	(* Internal method *)
	{attribute 'hide'}
	METHOD FB_init : BOOL
	VAR_INPUT
		(*  if TRUE, the retain variables are initialized (warm start / cold start) *)
		bInitRetains : BOOL;
		(*  if TRUE, the instance afterwards gets moved into the copy code (online change) *)
		bInCopyCode : BOOL;
	END_VAR
END_METHOD


	(* Internal method *)
	{attribute 'hide'}
	METHOD FB_exit : BOOL
	VAR_INPUT
		(*  if TRUE, the exit method is called for exiting an instance that is copied afterwards (online change). *)
		bInCopyCode : BOOL;
	END_VAR
END_METHOD


	(* Set the rotation angle in degrees [Â°]. *)
	METHOD SetAngle
	VAR_INPUT
		(* Rotation angle to set in degrees [Â°]. *)
		angle : LREAL;
	END_VAR
END_METHOD


	(* Set the components of this vector to '0.0'. *)
	METHOD SetZero
END_METHOD


	(* Set the components of this orientation. *)
	METHOD SetValues
	VAR_IN_OUT
		(* The position values to set. *)
 {attribute 'GUID' := '86B4AC92-A3FD-99C6-DFBE-A266E31A06E2'}
				orientation2D : Orientation2D;
	END_VAR
END_METHOD


	(* Get the direction of the local x-axis. *)
	METHOD GetDirectionX
	VAR_IN_OUT
		(* The local x-direction of this orientation. *)
 {attribute 'GUID' := '4CE6AEBB-A122-94B9-C485-29D927BD5C71'}
				localX : TangentXY;
	END_VAR
END_METHOD


	(* Get the direction of the local y-axis. *)
	METHOD GetDirectionY
	VAR_IN_OUT
		(* The local y-direction of this orientation. *)
 {attribute 'GUID' := '4CE6AEBB-A122-94B9-C485-29D927BD5C71'}
				localY : TangentXY;
	END_VAR
END_METHOD


	(* Invert this position. *)
	METHOD Invert
END_METHOD


	(* Multiply an orientation to this orientation. *)
	METHOD ConcatenateWith
	VAR_IN_OUT
		(* Orientation to concatenate with. *)
 {attribute 'GUID' := '86B4AC92-A3FD-99C6-DFBE-A266E31A06E2'}
				orientation2D : Orientation2D;
	END_VAR
END_METHOD


	(* Turn the orientation. *)
	METHOD TurnByC
	VAR_INPUT
		(* Rotation angle to turn by in degrees [Â°]. *)
		angle : LREAL;
	END_VAR
END_METHOD


	(* Rotate a PositionXY according to this orientation. *)
	METHOD Transform
	VAR_IN_OUT
		(* The orientation to multipy by. *)
 {attribute 'GUID' := 'FCACA74E-C57F-9E9F-C3FF-7BECD9A9CD0E'}
				positionXY : PositionXY;
	END_VAR
END_METHOD


	PROPERTY angle : LREAL
GET
END_GET
SET
END_SET
END_PROPERTY

END_FUNCTION_BLOCK

// POUs/Spatial/Functions/ConcatenateABC

	{attribute 'TcIecLibraryType'}
	{attribute 'external_name' := 'ConcatenateABC_GUID_72325069_8572_94A4_CBCD_8734C10F3E88'}
	(* Concatenate two instances of Orientation3D. *)
	FUNCTION ConcatenateABC : BOOL
	VAR_IN_OUT
		rotation0	:	Orientation3D;	(* 1st input orientation of the concatenation. *)
		rotation1	:	Orientation3D;	(* 2nd input orientation of the concatenation. *)
		concatenation	:	Orientation3D;	(* The concatenation of the two input instances. *)
	END_VAR

END_FUNCTION

// POUs/Spatial/Positions/Orientation3D

	{attribute 'c++_compatible'}
	{attribute 'external_name' := 'Orientation3D_GUID_E2786DA7_805D_90A4_CCD0_35D19D53662E'}
	{attribute 'TcIecLibraryType'}
	{attribute 'no_explicit_call' :='do not call this POU directly'}
	{attribute 'no_assign'}
	(* 3D orientation. All angles in degrees [Â°]. *)
	FUNCTION_BLOCK Orientation3D
	VAR
		(* Rotation around the 1st local axis in degrees [Â°]. *)
		p0 : LREAL;
		(* Rotation around 2nd local axis in degrees [Â°]. *)
		p1 : LREAL;
		(* Rotation around 3rd local axis in degrees [Â°]. *)
		p2 : LREAL;
		(* Defines the rotation order (rotate around local axes from left to right) *)
		 {attribute 'GUID' := 'BF8BCC1E-925E-4A57-801C-CC42AFDDA86D'}
		coordinates : E_RotationCoordinates := E_RotationCoordinates.CBA;
		 {attribute 'hide'}
		_reserved1 : ARRAY [1..84] OF USINT;
	END_VAR


	(* Internal method *)
	{attribute 'hide'}
	METHOD FB_init : BOOL
	VAR_INPUT
		(*  if TRUE, the retain variables are initialized (warm start / cold start) *)
		bInitRetains : BOOL;
		(*  if TRUE, the instance afterwards gets moved into the copy code (online change) *)
		bInCopyCode : BOOL;
	END_VAR
END_METHOD


	(* Internal method *)
	{attribute 'hide'}
	METHOD FB_exit : BOOL
	VAR_INPUT
		(*  if TRUE, the exit method is called for exiting an instance that is copied afterwards (online change). *)
		bInCopyCode : BOOL;
	END_VAR
END_METHOD


	(* Set the components of this vector to '0.0'. *)
	METHOD SetZero
END_METHOD


	(* Set the components of this position. *)
	METHOD SetValues
	VAR_IN_OUT
		(* The position values to set. *)
 {attribute 'GUID' := 'E2786DA7-805D-90A4-CCD0-35D19D53662E'}
				orientation3D : Orientation3D;
	END_VAR
END_METHOD


	(* Set the coordinates of the orientation. *)
	METHOD SetValuesABC
	VAR_INPUT
		(* 1st rotation angle in degrees [Â°]. *)
		phi0 : LREAL;
		(* 2nd rotation angle in degrees [Â°]. *)
		phi1 : LREAL;
		(* 3rd rotation angle in degrees [Â°]. *)
		phi2 : LREAL;
	END_VAR
END_METHOD


	(* Set the coordinates of the orientation. *)
	METHOD SetValuesACB
	VAR_INPUT
		(* 1st rotation angle in degrees [Â°]. *)
		phi0 : LREAL;
		(* 2nd rotation angle in degrees [Â°]. *)
		phi1 : LREAL;
		(* 3rd rotation angle in degrees [Â°]. *)
		phi2 : LREAL;
	END_VAR
END_METHOD


	(* Set the coordinates of the orientation. *)
	METHOD SetValuesBCA
	VAR_INPUT
		(* 1st rotation angle in degrees [Â°]. *)
		phi0 : LREAL;
		(* 2nd rotation angle in degrees [Â°]. *)
		phi1 : LREAL;
		(* 3rd rotation angle in degrees [Â°]. *)
		phi2 : LREAL;
	END_VAR
END_METHOD


	(* Set the coordinates of the orientation. *)
	METHOD SetValuesBAC
	VAR_INPUT
		(* 1st rotation angle in degrees [Â°]. *)
		phi0 : LREAL;
		(* 2nd rotation angle in degrees [Â°]. *)
		phi1 : LREAL;
		(* 3rd rotation angle in degrees [Â°]. *)
		phi2 : LREAL;
	END_VAR
END_METHOD


	(* Set the coordinates of the orientation. *)
	METHOD SetValuesCAB
	VAR_INPUT
		(* 1st rotation angle in degrees [Â°]. *)
		phi0 : LREAL;
		(* 2nd rotation angle in degrees [Â°]. *)
		phi1 : LREAL;
		(* 3rd rotation angle in degrees [Â°]. *)
		phi2 : LREAL;
	END_VAR
END_METHOD


	(* Set the coordinates of the orientation. *)
	METHOD SetValuesCBA
	VAR_INPUT
		(* 1st rotation angle in degrees [Â°]. *)
		phi0 : LREAL;
		(* 2nd rotation angle in degrees [Â°]. *)
		phi1 : LREAL;
		(* 3rd rotation angle in degrees [Â°]. *)
		phi2 : LREAL;
	END_VAR
END_METHOD


	(* Set the coordinates of the orientation. *)
	METHOD SetValuesABA
	VAR_INPUT
		(* 1st rotation angle in degrees [Â°]. *)
		phi0 : LREAL;
		(* 2nd rotation angle in degrees [Â°]. *)
		phi1 : LREAL;
		(* 3rd rotation angle in degrees [Â°]. *)
		phi2 : LREAL;
	END_VAR
END_METHOD


	(* Set the coordinates of the orientation. *)
	METHOD SetValuesACA
	VAR_INPUT
		(* 1st rotation angle in degrees [Â°]. *)
		phi0 : LREAL;
		(* 2nd rotation angle in degrees [Â°]. *)
		phi1 : LREAL;
		(* 3rd rotation angle in degrees [Â°]. *)
		phi2 : LREAL;
	END_VAR
END_METHOD


	(* Set the coordinates of the orientation. *)
	METHOD SetValuesBCB
	VAR_INPUT
		(* 1st rotation angle in degrees [Â°]. *)
		phi0 : LREAL;
		(* 2nd rotation angle in degrees [Â°]. *)
		phi1 : LREAL;
		(* 3rd rotation angle in degrees [Â°]. *)
		phi2 : LREAL;
	END_VAR
END_METHOD


	(* Set the coordinates of the orientation. *)
	METHOD SetValuesBAB
	VAR_INPUT
		(* 1st rotation angle in degrees [Â°]. *)
		phi0 : LREAL;
		(* 2nd rotation angle in degrees [Â°]. *)
		phi1 : LREAL;
		(* 3rd rotation angle in degrees [Â°]. *)
		phi2 : LREAL;
	END_VAR
END_METHOD


	(* Set the coordinates of the orientation. *)
	METHOD SetValuesCAC
	VAR_INPUT
		(* 1st rotation angle in degrees [Â°]. *)
		phi0 : LREAL;
		(* 2nd rotation angle in degrees [Â°]. *)
		phi1 : LREAL;
		(* 3rd rotation angle in degrees [Â°]. *)
		phi2 : LREAL;
	END_VAR
END_METHOD


	(* Set the coordinates of the orientation. *)
	METHOD SetValuesCBC
	VAR_INPUT
		(* 1st rotation angle in degrees [Â°]. *)
		phi0 : LREAL;
		(* 2nd rotation angle in degrees [Â°]. *)
		phi1 : LREAL;
		(* 3rd rotation angle in degrees [Â°]. *)
		phi2 : LREAL;
	END_VAR
END_METHOD


	(* Get the direction of the local x-axis. *)
	METHOD GetDirectionX
	VAR_IN_OUT
		(* The local x-direction of this orientation. *)
 {attribute 'GUID' := '9F987066-55C3-9A71-FEA1-9CB49A451CD6'}
				localX : Tangent3D;
	END_VAR
END_METHOD


	(* Get the direction of the local y-axis. *)
	METHOD GetDirectionY
	VAR_IN_OUT
		(* The local y-direction of this orientation. *)
 {attribute 'GUID' := '9F987066-55C3-9A71-FEA1-9CB49A451CD6'}
				localY : Tangent3D;
	END_VAR
END_METHOD


	(* Get the direction of the local z-axis. *)
	METHOD GetDirectionZ
	VAR_IN_OUT
		(* The local z-direction of this orientation. *)
 {attribute 'GUID' := '9F987066-55C3-9A71-FEA1-9CB49A451CD6'}
				localZ : Tangent3D;
	END_VAR
END_METHOD


	(* Invert this position. *)
	METHOD Invert
END_METHOD


	(* Multiply an orientation to this orientation. *)
	METHOD ConcatenateWith
	VAR_IN_OUT
		(* Orientation to concatenate with. *)
 {attribute 'GUID' := 'E2786DA7-805D-90A4-CCD0-35D19D53662E'}
				orientation : Orientation3D;
	END_VAR
END_METHOD


	(* Rotate around an arbitrary local axis. The turn angle is given by the length of the axis. *)
	METHOD TurnBy
	VAR_IN_OUT
		(* The axis of rotation. Its length represents the angle of rotation in degrees [Â°]. *)
 {attribute 'GUID' := '6DC08058-799F-98C7-C4DD-73FA46FCF197'}
				axis : TangentABC;
	END_VAR
END_METHOD


	(* Rotation around the local x-axis. *)
	METHOD TurnByA
	VAR_INPUT
		(* The angle to rotate by in degrees [Â°]. *)
		da : LREAL;
	END_VAR
END_METHOD


	(* Rotation around the local y-axis. *)
	METHOD TurnByB
	VAR_INPUT
		(* The angle to rotate by in degrees [Â°]. *)
		db : LREAL;
	END_VAR
END_METHOD


	(* Rotation around the local z-axis. *)
	METHOD TurnByC
	VAR_INPUT
		(* The angle to rotate by in degrees [Â°]. *)
		dc : LREAL;
	END_VAR
END_METHOD


	(* Rotate a Position3D according to this orientation. *)
	METHOD Transform
	VAR_IN_OUT
		(* Position to transform. *)
 {attribute 'GUID' := '40E6105C-AAE1-907F-E93C-27FE8D6C7544'}
				position3D : Position3D;
	END_VAR
END_METHOD


	PROPERTY phi0 : LREAL
GET
END_GET
SET
END_SET
END_PROPERTY


	PROPERTY phi1 : LREAL
GET
END_GET
SET
END_SET
END_PROPERTY


	PROPERTY phi2 : LREAL
GET
END_GET
SET
END_SET
END_PROPERTY


	PROPERTY convention : E_RotationCoordinates
GET
END_GET
SET
END_SET
END_PROPERTY

END_FUNCTION_BLOCK

// POUs/Spatial/Functions/ConcatenateXYC

	{attribute 'TcIecLibraryType'}
	{attribute 'external_name' := 'ConcatenateXYC_GUID_55AD0630_DF53_9402_CBF6_9E8FF05A606D'}
	(* Concatenate two instances of PositionXYC. *)
	FUNCTION ConcatenateXYC : BOOL
	VAR_IN_OUT
		position0	:	PositionXYC;	(* 1st input position of the concatenation. *)
		position1	:	PositionXYC;	(* 2nd input position of the concatenation. *)
		concatenation	:	PositionXYC;	(* The concatenation of the two input instances. *)
	END_VAR

END_FUNCTION

// POUs/Spatial/Functions/Concatenate6D

	{attribute 'TcIecLibraryType'}
	{attribute 'external_name' := 'Concatenate6D_GUID_A3C51CBA_D129_9074_F963_7F4312C3BE5C'}
	(* Concatenate two instances of PositionSE3. *)
	FUNCTION Concatenate6D : BOOL
	VAR_IN_OUT
		position0	:	PositionSE3;	(* 1st input position of the concatenation. *)
		position1	:	PositionSE3;	(* 2nd input position of the concatenation. *)
		concatenation	:	PositionXYC;	(* The concatenation of the two input instances. *)
	END_VAR

END_FUNCTION

// POUs/Spatial/Functions/AddXY

	{attribute 'TcIecLibraryType'}
	{attribute 'external_name' := 'AddXY_GUID_F0A8AB4F_2A83_9A21_FF35_C9D3AB4C34D2'}
	(* Add two instances of TangentXY. *)
	FUNCTION AddXY : BOOL
	VAR_IN_OUT
		tangent0	:	TangentXY;	(* 1st input tangent vector. *)
		tangent1	:	TangentXY;	(* 2nd input tangent vector. *)
		sumTangent	:	TangentXY;	(* Sum of the two tangent vectors. *)
	END_VAR

END_FUNCTION

// POUs/Spatial/Functions/SubtractXY

	{attribute 'TcIecLibraryType'}
	{attribute 'external_name' := 'SubtractXY_GUID_2114A8BE_2197_98FB_CE09_32138D555625'}
	(* Subtract two instances of TangentXY. *)
	FUNCTION SubtractXY : BOOL
	VAR_IN_OUT
		tangent0	:	TangentXY;	(* 1st input tangent vector. *)
		tangent1	:	TangentXY;	(* 2nd input tangent vector. *)
		difference	:	TangentXY;	(* Difference of the two tangent vectors. *)
	END_VAR

END_FUNCTION

// POUs/Spatial/Functions/MultiplyXY

	{attribute 'TcIecLibraryType'}
	{attribute 'external_name' := 'MultiplyXY_GUID_EFBF5EAA_3662_985E_C980_B34A9211CE75'}
	(* Multiply a TangentXY by a scalar and return the result. *)
	FUNCTION MultiplyXY : BOOL
	VAR_IN_OUT
		tangent	:	TangentXY;	(* Tangent vector to multiply. *)
	END_VAR
	VAR_INPUT
		scalar	:	LREAL;	(* Scalar value to multiply with. *)
	END_VAR
	VAR_IN_OUT
		scaled	:	TangentXY;	(* Scaled input tangent vector. *)
	END_VAR

END_FUNCTION

// POUs/Spatial/Functions/ScalarXY

	{attribute 'TcIecLibraryType'}
	{attribute 'external_name' := 'ScalarXY_GUID_F9A29ED6_D852_9E87_C12A_8471B8CCADB2'}
	(* Compute the scalar product of two instance of TangentXY. *)
	FUNCTION ScalarXY : LREAL
	VAR_IN_OUT
		tangent0	:	TangentXY;	(* 1st input tangent vector. *)
		tangent1	:	TangentXY;	(* 2nd input tangent vector. *)
	END_VAR

END_FUNCTION

// POUs/Spatial/Functions/Add3D

	{attribute 'TcIecLibraryType'}
	{attribute 'external_name' := 'Add3D_GUID_33681FAC_919A_96DC_E61A_A0C04831E109'}
	(* Add two instances of Tangent3D. *)
	FUNCTION Add3D : BOOL
	VAR_IN_OUT
		tangent0	:	Tangent3D;	(* 1st input tangent vector. *)
		tangent1	:	Tangent3D;	(* 2nd input tangent vector. *)
		sumTangent	:	Tangent3D;	(* Sum of the two tangent vectors. *)
	END_VAR

END_FUNCTION

// POUs/Spatial/Functions/Subtract3D

	{attribute 'TcIecLibraryType'}
	{attribute 'external_name' := 'Subtract3D_GUID_2ECEB7F8_2A80_9372_C8D0_F4C330030BDB'}
	(* Subtract two instances of Tangent3D. *)
	FUNCTION Subtract3D : BOOL
	VAR_IN_OUT
		tangent0	:	Tangent3D;	(* 1st input tangent vector. *)
		tangent1	:	Tangent3D;	(* 2nd input tangent vector. *)
		difference	:	Tangent3D;	(* Difference of the two tangent vectors. *)
	END_VAR

END_FUNCTION

// POUs/Spatial/Functions/Multiply3D

	{attribute 'TcIecLibraryType'}
	{attribute 'external_name' := 'Multiply3D_GUID_526B136B_20EA_972E_C6AE_56E6AECFFFD9'}
	(* Multiply a Tangent3D by a scalar. *)
	FUNCTION Multiply3D : BOOL
	VAR_IN_OUT
		tangent	:	Tangent3D;	(* Tangent vector to multiply. *)
	END_VAR
	VAR_INPUT
		scalar	:	LREAL;	(* Scalar value to multiply with. *)
	END_VAR
	VAR_IN_OUT
		scaled	:	Tangent3D;	(* Scaled input tangent vector. *)
	END_VAR

END_FUNCTION

// POUs/Spatial/Functions/Scalar3D

	{attribute 'TcIecLibraryType'}
	{attribute 'external_name' := 'Scalar3D_GUID_A78BB39E_7D88_9437_DBE7_D1F64786C431'}
	(* Compute the scalar product of two instances of Tangent3D. *)
	FUNCTION Scalar3D : LREAL
	VAR_IN_OUT
		tangent0	:	Tangent3D;	(* 1st input tangent vector. *)
		tangent1	:	Tangent3D;	(* 2nd input tangent vector. *)
	END_VAR

END_FUNCTION

// POUs/Spatial/Functions/Cross3D

	{attribute 'TcIecLibraryType'}
	{attribute 'external_name' := 'Cross3D_GUID_72A34119_3753_97FA_E3C4_99EE49EDB00C'}
	(* Compute the cross product of two instances of Tangent3D. *)
	FUNCTION Cross3D : BOOL
	VAR_IN_OUT
		tangent0	:	Tangent3D;	(* 1st input tangent vector. *)
		tangent1	:	Tangent3D;	(* 2nd input tangent vector. *)
		crossProduct	:	Tangent3D;	(* The resulting cross product. *)
	END_VAR

END_FUNCTION

// POUs/Spatial/Functions/AddABC

	{attribute 'TcIecLibraryType'}
	{attribute 'external_name' := 'AddABC_GUID_A2A585C2_9704_99E4_F95C_2BFAFA04D5A7'}
	(* Add two instances of TangentABC. *)
	FUNCTION AddABC : BOOL
	VAR_IN_OUT
		tangent0	:	TangentABC;	(* 1st input tangent vector. *)
		tangent1	:	TangentABC;	(* 2nd input tangent vector. *)
		sumTangent	:	TangentABC;	(* Sum of the two tangent vectors. *)
	END_VAR

END_FUNCTION

// POUs/Spatial/Functions/SubtractABC

	{attribute 'TcIecLibraryType'}
	{attribute 'external_name' := 'SubtractABC_GUID_1F1A1DC3_BCE2_9B37_CCA9_1A20F5CCE622'}
	(* Subtract two instances of TangentABC. *)
	FUNCTION SubtractABC : BOOL
	VAR_IN_OUT
		tangent0	:	TangentABC;	(* 1st input tangent vector. *)
		tangent1	:	TangentABC;	(* 2nd input tangent vector. *)
		difference	:	TangentABC;	(* Difference of the two tangent vectors. *)
	END_VAR

END_FUNCTION

// POUs/Spatial/Functions/MultiplyABC

	{attribute 'TcIecLibraryType'}
	{attribute 'external_name' := 'MultiplyABC_GUID_DF081CCC_423C_9472_DB33_1877A6381F0C'}
	(* Multiply a TangentABC by a scalar. *)
	FUNCTION MultiplyABC : BOOL
	VAR_IN_OUT
		tangent	:	TangentABC;	(* Tangent vector to multiply. *)
	END_VAR
	VAR_INPUT
		scalar	:	LREAL;	(* Scalar value to multiply with. *)
	END_VAR
	VAR_IN_OUT
		scaled	:	TangentABC;	(* Scaled input tangent vector. *)
	END_VAR

END_FUNCTION

// POUs/Spatial/Functions/AddXYC

	{attribute 'TcIecLibraryType'}
	{attribute 'external_name' := 'AddXYC_GUID_0FC928B9_D3BF_9FE8_C6B0_572CE1F84885'}
	(* Add two instances of TangentXYC. *)
	FUNCTION AddXYC : BOOL
	VAR_IN_OUT
		tangent0	:	TangentXYC;	(* 1st input tangent vector. *)
		tangent1	:	TangentXYC;	(* 2nd input tangent vector. *)
		sumTangent	:	TangentXYC;	(* Sum of the two tangent vectors. *)
	END_VAR

END_FUNCTION

// POUs/Spatial/Functions/SubtractXYC

	{attribute 'TcIecLibraryType'}
	{attribute 'external_name' := 'SubtractXYC_GUID_CC347E26_8071_91B2_F9A5_D41F53C922C2'}
	(* Subtract two instances of TangentXYC. *)
	FUNCTION SubtractXYC : BOOL
	VAR_IN_OUT
		tangent0	:	TangentXYC;	(* 1st input tangent vector. *)
		tangent1	:	TangentXYC;	(* 2nd input tangent vector. *)
		difference	:	TangentXYC;	(* Difference of the two tangent vectors. *)
	END_VAR

END_FUNCTION

// POUs/Spatial/Functions/MultiplyXYC

	{attribute 'TcIecLibraryType'}
	{attribute 'external_name' := 'MultiplyXYC_GUID_7AEEEA34_80B2_9AC1_FC91_2F8A3AE52498'}
	(* Multiply a TangentXYC by a scalar. *)
	FUNCTION MultiplyXYC : BOOL
	VAR_IN_OUT
		tangent	:	TangentXYC;	(* Tangent vector to multiply. *)
	END_VAR
	VAR_INPUT
		scalar	:	LREAL;	(* Scalar value to multiply with. *)
	END_VAR
	VAR_IN_OUT
		scaled	:	TangentXYC;	(* Scaled input tangent vector. *)
	END_VAR

END_FUNCTION

// POUs/Spatial/Functions/Add6D

	{attribute 'TcIecLibraryType'}
	{attribute 'external_name' := 'Add6D_GUID_1AC97E8A_D619_93C4_CB56_5792DE8B457A'}
	(* Add two instances of Tangent6D. *)
	FUNCTION Add6D : BOOL
	VAR_IN_OUT
		tangent0	:	Tangent6D;	(* 1st input tangent vector. *)
		tangent1	:	Tangent6D;	(* 2nd input tangent vector. *)
		sumTangent	:	Tangent6D;	(* Sum of the two tangent vectors. *)
	END_VAR

END_FUNCTION

// POUs/Spatial/Functions/Subtract6D

	{attribute 'TcIecLibraryType'}
	{attribute 'external_name' := 'Subtract6D_GUID_EF5A0440_CB1C_9C2B_EE25_AA331DF61931'}
	(* Subtract two instances of Tangent6D. *)
	FUNCTION Subtract6D : BOOL
	VAR_IN_OUT
		tangent0	:	Tangent6D;	(* 1st input tangent vector. *)
		tangent1	:	Tangent6D;	(* 2nd input tangent vector. *)
		difference	:	Tangent6D;	(* Difference of the two tangent vectors. *)
	END_VAR

END_FUNCTION

// POUs/Spatial/Functions/Multiply6D

	{attribute 'TcIecLibraryType'}
	{attribute 'external_name' := 'Multiply6D_GUID_FB076CD1_A9A2_9FC6_F4A8_5EADCA86AB35'}
	(* Multiply a Tangent6D by a scalar. *)
	FUNCTION Multiply6D : BOOL
	VAR_IN_OUT
		tangent	:	Tangent6D;	(* Tangent vector to multiply. *)
	END_VAR
	VAR_INPUT
		scalar	:	LREAL;	(* Scalar value to multiply with. *)
	END_VAR
	VAR_IN_OUT
		scaled	:	Tangent6D;	(* Scaled input tangent vector. *)
	END_VAR

END_FUNCTION

// POUs/Spatial/Functions/ConvertToCartesian2D

	{attribute 'TcIecLibraryType'}
	{attribute 'external_name' := 'ConvertToCartesian2D_GUID_77BE389F_A1A9_96B4_CB70_469C2431A8D6'}
	(* Convert local XYC-dynamic properties to global XY ones. *)
	FUNCTION ConvertToCartesian2D : BOOL
	VAR_IN_OUT
		position	:	PositionXYC;	(* The position hosting the local dynamic state. *)
		velocity	:	TangentXYC;	(* The local velocity vector. *)
		acceleration	:	TangentXYC;	(* The local acceleration vector. *)
		velocity_XY	:	TangentXY;	(* The resulting global Cartesian velocity. *)
		acceleration_XY	:	TangentXY;	(* The resulting global Cartesian acceleration. *)
	END_VAR

END_FUNCTION

// POUs/Spatial/Setpoints/SetpointR1

	{attribute 'c++_compatible'}
	{attribute 'external_name' := 'SetpointR1_GUID_26A6180F_A0FD_9529_FBAE_6B2E931D373F'}
	{attribute 'TcIecLibraryType'}
	{attribute 'no_explicit_call' :='do not call this POU directly'}
	{attribute 'no_assign_warning'}
	(* 1D setpoint. *)
	FUNCTION_BLOCK SetpointR1
	VAR
		(* Position component of the setpoint. *)
		ds : LREAL;
		(* Velocity component of the setpoint. *)
		dv : LREAL;
		(* Acceleration component of the setpoint. *)
		da : LREAL;
		(* Jerk component of the setpoint. *)
		dj : LREAL;
	END_VAR


	(* Internal method *)
	{attribute 'hide'}
	METHOD FB_init : BOOL
	VAR_INPUT
		(*  if TRUE, the retain variables are initialized (warm start / cold start) *)
		bInitRetains : BOOL;
		(*  if TRUE, the instance afterwards gets moved into the copy code (online change) *)
		bInCopyCode : BOOL;
	END_VAR
END_METHOD


	(* Internal method *)
	{attribute 'hide'}
	METHOD FB_reinit : BOOL
END_METHOD


	(* Internal method *)
	{attribute 'hide'}
	METHOD FB_exit : BOOL
	VAR_INPUT
		(*  if TRUE, the exit method is called for exiting an instance that is copied afterwards (online change). *)
		bInCopyCode : BOOL;
	END_VAR
END_METHOD


	(* Set this setpoint to zero. *)
	METHOD SetZero
END_METHOD


	(* Set the values of this coordinate. *)
	METHOD SetValuesSVAJ
	VAR_INPUT
		(* the position value to set. *)
		_s : LREAL;
		(* the velocity value to set. *)
		v : LREAL;
		(* the acceleration value to set. *)
		a : LREAL;
		(* the jerk value to set. *)
		j : LREAL;
	END_VAR
END_METHOD


	PROPERTY _s : LREAL
GET
END_GET
SET
END_SET
END_PROPERTY


	PROPERTY v : LREAL
GET
END_GET
SET
END_SET
END_PROPERTY


	PROPERTY a : LREAL
GET
END_GET
SET
END_SET
END_PROPERTY


	PROPERTY j : LREAL
GET
END_GET
SET
END_SET
END_PROPERTY

END_FUNCTION_BLOCK

// POUs/Spatial/Setpoints/SetpointSE3

	{attribute 'c++_compatible'}
	{attribute 'external_name' := 'SetpointSE3_GUID_B229B847_5FB0_9D40_DB46_E3FDC33C7140'}
	{attribute 'TcIecLibraryType'}
	{attribute 'no_explicit_call' :='do not call this POU directly'}
	{attribute 'no_assign_warning'}
	(* SE3 setpoint. *)
	FUNCTION_BLOCK SetpointSE3 EXTENDS IPlcGeometry3D


	(* Internal method *)
	{attribute 'hide'}
	METHOD FB_init : BOOL
	VAR_INPUT
		(*  if TRUE, the retain variables are initialized (warm start / cold start) *)
		bInitRetains : BOOL;
		(*  if TRUE, the instance afterwards gets moved into the copy code (online change) *)
		bInCopyCode : BOOL;
	END_VAR
END_METHOD


	(* Internal method *)
	{attribute 'hide'}
	METHOD FB_exit : BOOL
	VAR_INPUT
		(*  if TRUE, the exit method is called for exiting an instance that is copied afterwards (online change). *)
		bInCopyCode : BOOL;
	END_VAR
END_METHOD


	(* Set this setpoint to be the identity. *)
	METHOD SetIdentity
END_METHOD


	(* Set the values of this setpoint. *)
	METHOD SetValues
	VAR_IN_OUT
		(* The setpoint to copy. *)
 {attribute 'GUID' := 'B229B847-5FB0-9D40-DB46-E3FDC33C7140'}
				setpoint : SetpointSE3;
	END_VAR
END_METHOD


	(* Set the cartesian values of this setpoint. *)
	METHOD SetValuesXYZ
	VAR_IN_OUT
		(* The x-setpoint to set. *)
 {attribute 'GUID' := '26A6180F-A0FD-9529-FBAE-6B2E931D373F'}
				setpointX : SetpointR1;
		(* The y-setpoint to set. *)
 {attribute 'GUID' := '26A6180F-A0FD-9529-FBAE-6B2E931D373F'}
				setpointY : SetpointR1;
		(* The z-setpoint to set. *)
 {attribute 'GUID' := '26A6180F-A0FD-9529-FBAE-6B2E931D373F'}
				setpointZ : SetpointR1;
	END_VAR
END_METHOD


	(* Set the angular values of this setpoint. *)
	METHOD SetValuesCBA
	VAR_IN_OUT
		(* The c-setpoint to set. *)
 {attribute 'GUID' := '26A6180F-A0FD-9529-FBAE-6B2E931D373F'}
				setpointC : SetpointR1;
		(* The b-setpoint to set. *)
 {attribute 'GUID' := '26A6180F-A0FD-9529-FBAE-6B2E931D373F'}
				setpointB : SetpointR1;
		(* The a-setpoint to set. *)
 {attribute 'GUID' := '26A6180F-A0FD-9529-FBAE-6B2E931D373F'}
				setpointA : SetpointR1;
	END_VAR
END_METHOD


	(* Get the direction of the local x-axis. *)
	METHOD GetDirectionX
	VAR_IN_OUT
		(* The local x-direction of this orientation. *)
 {attribute 'GUID' := '9F987066-55C3-9A71-FEA1-9CB49A451CD6'}
				localX : Tangent3D;
	END_VAR
END_METHOD


	(* Get the direction of the local y-axis. *)
	METHOD GetDirectionY
	VAR_IN_OUT
		(* The local y-direction of this orientation. *)
 {attribute 'GUID' := '9F987066-55C3-9A71-FEA1-9CB49A451CD6'}
				localY : Tangent3D;
	END_VAR
END_METHOD


	(* Get the direction of the local z-axis. *)
	METHOD GetDirectionZ
	VAR_IN_OUT
		(* The local z-direction of this orientation. *)
 {attribute 'GUID' := '9F987066-55C3-9A71-FEA1-9CB49A451CD6'}
				localZ : Tangent3D;
	END_VAR
END_METHOD


	(* Get the linear Cartesian position components. *)
	METHOD GetPosition_Cartesian
	VAR_IN_OUT
		(* The output position. *)
 {attribute 'GUID' := '40E6105C-AAE1-907F-E93C-27FE8D6C7544'}
				position : Position3D;
	END_VAR
END_METHOD


	(* Get the linear Cartesian velocity components. *)
	METHOD GetVelocity_Cartesian
	VAR_IN_OUT
		(* The output tangent. *)
 {attribute 'GUID' := '9F987066-55C3-9A71-FEA1-9CB49A451CD6'}
				tangent : Tangent3D;
	END_VAR
END_METHOD


	(* Get the linear Cartesian acceleration components. *)
	METHOD GetAcceleration_Cartesian
	VAR_IN_OUT
		(* The output tangent. *)
 {attribute 'GUID' := '9F987066-55C3-9A71-FEA1-9CB49A451CD6'}
				tangent : Tangent3D;
	END_VAR
END_METHOD


	(* Get the linear Cartesian jerk components. *)
	METHOD GetJerk_Cartesian
	VAR_IN_OUT
		(* The output tangent. *)
 {attribute 'GUID' := '9F987066-55C3-9A71-FEA1-9CB49A451CD6'}
				tangent : Tangent3D;
	END_VAR
END_METHOD


	(* Concatenate this setpoint with a second one up to a specific order. *)
	METHOD ConcatenateWith
	VAR_IN_OUT
		(* The setpoint to concatenate. *)
 {attribute 'GUID' := 'B229B847-5FB0-9D40-DB46-E3FDC33C7140'}
				setpoint : SetpointSE3;
	END_VAR
	VAR_INPUT
		(*  The order up to which to compute. *)
		order : UDINT;
	END_VAR
END_METHOD


	PROPERTY x : LREAL
GET
END_GET
SET
END_SET
END_PROPERTY


	PROPERTY y : LREAL
GET
END_GET
SET
END_SET
END_PROPERTY


	PROPERTY z : LREAL
GET
END_GET
SET
END_SET
END_PROPERTY


	PROPERTY phi0 : LREAL
GET
END_GET
SET
END_SET
END_PROPERTY


	PROPERTY phi1 : LREAL
GET
END_GET
SET
END_SET
END_PROPERTY


	PROPERTY phi2 : LREAL
GET
END_GET
SET
END_SET
END_PROPERTY


	PROPERTY Convention : E_RotationCoordinates
GET
END_GET
SET
END_SET
END_PROPERTY

END_FUNCTION_BLOCK

// POUs/Spatial/Inertias/InertiaSE3

	{attribute 'c++_compatible'}
	{attribute 'external_name' := 'InertiaSE3_GUID_2A78B02A_86B5_94F2_F4F8_8DBAF2850FC5'}
	{attribute 'TcIecLibraryType'}
	{attribute 'no_explicit_call' :='do not call this POU directly'}
	{attribute 'no_assign'}
	(* Inertia tensor containing angular and linear inertia. *)
	FUNCTION_BLOCK InertiaSE3
	VAR
		(* Mass of the inertia. *)
		m : LREAL;
		(* x-component of the center of mass. *)
		CenterX : LREAL;
		(* y-component of the center of mass. *)
		CenterY : LREAL;
		(* z-component of the center of mass. *)
		CenterZ : LREAL;
		 {attribute 'hide'}
		_reserved1 : ARRAY [1..80] OF USINT;
	END_VAR


	(* Internal method *)
	{attribute 'hide'}
	METHOD FB_init : BOOL
	VAR_INPUT
		(*  if TRUE, the retain variables are initialized (warm start / cold start) *)
		bInitRetains : BOOL;
		(*  if TRUE, the instance afterwards gets moved into the copy code (online change) *)
		bInCopyCode : BOOL;
	END_VAR
END_METHOD


	(* Internal method *)
	{attribute 'hide'}
	METHOD FB_exit : BOOL
	VAR_INPUT
		(*  if TRUE, the exit method is called for exiting an instance that is copied afterwards (online change). *)
		bInCopyCode : BOOL;
	END_VAR
END_METHOD


	(* Add a 2nd inertia tensor to this one. *)
	METHOD AddBy
	VAR_IN_OUT
		(* The inertia tensor to add. *)
 {attribute 'GUID' := '2A78B02A-86B5-94F2-F4F8-8DBAF2850FC5'}
				shift : InertiaSE3;
	END_VAR
END_METHOD


	(* Set the values to that of a point. *)
	METHOD SetValues_Point
	VAR_INPUT
		(* The mass of the point. *)
		mass : LREAL;
		(* The x-position of the point. *)
		x : LREAL;
		(* The y-position of the point. *)
		y : LREAL;
		(* The z-position of the point. *)
		z : LREAL;
	END_VAR
END_METHOD


	(* Set the values to that of a sphere. *)
	METHOD SetValues_Sphere
	VAR_INPUT
		(* The mass of the sphere. *)
		mass : LREAL;
		(* The radius of the sphere. *)
		radius : LREAL;
	END_VAR
END_METHOD


	(* Set the values to that of a cylinder. *)
	METHOD SetValues_Cylinder
	VAR_INPUT
		(* The mass of the cylinder. *)
		mass : LREAL;
		(* The radius of the cylinder. *)
		radius : LREAL;
		(* The height of the cylinder. *)
		height : LREAL;
	END_VAR
END_METHOD


	(* Set the values to that of a cuboid. *)
	METHOD SetValues_Cuboid
	VAR_INPUT
		(* The mass of the cuboid. *)
		mass : LREAL;
		(* The x-length of the cuboid. *)
		dx : LREAL;
		(* The y-length of the cuboid. *)
		dy : LREAL;
		(* The z-length of the cuboid. *)
		dz : LREAL;
	END_VAR
END_METHOD


	(* Transform this inertia by a displacement. *)
	METHOD Transform
	VAR_IN_OUT
		(* The displacement to apply. *)
 {attribute 'GUID' := '608A620D-3BBF-9A33-F5CB-39FFBA2AADD1'}
				displacement : PositionSE3;
	END_VAR
END_METHOD


	(* Translate this inertia by a translation. *)
	METHOD Translate
	VAR_IN_OUT
		(* The translation to apply. *)
 {attribute 'GUID' := '9F987066-55C3-9A71-FEA1-9CB49A451CD6'}
				displacement : Tangent3D;
	END_VAR
END_METHOD


	PROPERTY mass : LREAL
GET
END_GET
SET
END_SET
END_PROPERTY


	PROPERTY x : LREAL
GET
END_GET
SET
END_SET
END_PROPERTY


	PROPERTY y : LREAL
GET
END_GET
SET
END_SET
END_PROPERTY


	PROPERTY z : LREAL
GET
END_GET
SET
END_SET
END_PROPERTY


	PROPERTY xx : LREAL
GET
END_GET
SET
END_SET
END_PROPERTY


	PROPERTY yy : LREAL
GET
END_GET
SET
END_SET
END_PROPERTY


	PROPERTY zz : LREAL
GET
END_GET
SET
END_SET
END_PROPERTY


	PROPERTY xy : LREAL
GET
END_GET
SET
END_SET
END_PROPERTY


	PROPERTY yz : LREAL
GET
END_GET
SET
END_SET
END_PROPERTY


	PROPERTY zx : LREAL
GET
END_GET
SET
END_SET
END_PROPERTY

END_FUNCTION_BLOCK

// POUs/Shapes/Geometry2D/Container2D

	{attribute 'c++_compatible'}
	{attribute 'external_name' := 'Container2D_GUID_5B056115_040C_99AB_F38A_306B253376A0'}
	{attribute 'TcIecLibraryType'}
	{attribute 'no_explicit_call' :='do not call this POU directly'}
	{attribute 'no_assign'}
	FUNCTION_BLOCK Container2D EXTENDS Geometry2D


	(* Internal method *)
	METHOD FB_init : BOOL
	VAR_INPUT
		(*  if TRUE, the retain variables are initialized (warm start / cold start) *)
		bInitRetains : BOOL;
		(*  if TRUE, the instance afterwards gets moved into the copy code (online change) *)
		bInCopyCode : BOOL;
	END_VAR
END_METHOD


	(* Internal method *)
	{attribute 'hide'}
	METHOD FB_exit : BOOL
	VAR_INPUT
		(*  if TRUE, the exit method is called for exiting an instance that is copied afterwards (online change). *)
		bInCopyCode : BOOL;
	END_VAR
END_METHOD


	(* Add a geometry to the container. *)
	METHOD AddElement : UDINT
	VAR_IN_OUT
		(* The geometry to add. *)
 {attribute 'GUID' := 'C762D668-D7C9-90ED-D0FC-88133F9DE94D'}
				inputObject : Geometry2D;
	END_VAR
END_METHOD


	(* Remove a specified geometry from the container. *)
	METHOD RemoveElement
	VAR_INPUT
		(* ID of the geometry to remove. *)
		id : UDINT;
	END_VAR
END_METHOD


	(* Remove all geometries from the container. *)
	METHOD Clear
END_METHOD


	(* Get the number of geometry elements in container. *)
	METHOD GetCount : UDINT
END_METHOD


	(* Get the combined boundary of all hosted 2D-geometries. *)
	METHOD GetBoundary
	VAR_IN_OUT
		(* The combined boundary.. *)
 {attribute 'GUID' := '5B056115-040C-99AB-F38A-306B253376A0'}
				boundary : Container2D;
	END_VAR
END_METHOD

END_FUNCTION_BLOCK

// POUs/Shapes/Geometry2D/Extrude2D

	{attribute 'c++_compatible'}
	{attribute 'external_name' := 'Extrude2D_GUID_CD67E7BE_FF79_9A12_FD80_AC96B1D32269'}
	{attribute 'TcIecLibraryType'}
	{attribute 'no_explicit_call' :='do not call this POU directly'}
	{attribute 'no_assign'}
	FUNCTION_BLOCK Extrude2D EXTENDS Geometry2D


	(* Internal method *)
	METHOD FB_init : BOOL
	VAR_INPUT
		(*  if TRUE, the retain variables are initialized (warm start / cold start) *)
		bInitRetains : BOOL;
		(*  if TRUE, the instance afterwards gets moved into the copy code (online change) *)
		bInCopyCode : BOOL;
	END_VAR
END_METHOD


	(* Internal method *)
	{attribute 'hide'}
	METHOD FB_exit : BOOL
	VAR_INPUT
		(*  if TRUE, the exit method is called for exiting an instance that is copied afterwards (online change). *)
		bInCopyCode : BOOL;
	END_VAR
END_METHOD


	(* Define the extrusion geometry by a path and the corners to extrude. *)
	METHOD ExtrudeAlong
	VAR_IN_OUT
		(* The path to extrude along. *)
 {attribute 'GUID' := '6E12F92E-6BF9-9AF0-D560-BBDFBB18383E'}
				path : PathXYC;
	END_VAR
	VAR_INPUT
		(* 1st distance from the path to extrude. *)
		dy0 : LREAL;
		(* 2nd distance from the path to extrude. *)
		dy1 : LREAL;
		(* Number of steps to employ along the path. *)
		extrusionSteps : UDINT;
	END_VAR
END_METHOD


	(* Check whether this extrusion geometry is valid. *)
	METHOD IsValid : BOOL
END_METHOD

END_FUNCTION_BLOCK

// POUs/Paths/Components/PathXYC

	{attribute 'c++_compatible'}
	{attribute 'external_name' := 'PathXYC_GUID_6E12F92E_6BF9_9AF0_D560_BBDFBB18383E'}
	{attribute 'TcIecLibraryType'}
	{attribute 'no_explicit_call' :='do not call this POU directly'}
	{attribute 'no_assign'}
	(* A path in the xy-plane with an additional orientation at every path position. *)
	FUNCTION_BLOCK PathXYC EXTENDS IPlcPath2D


	(* Internal method *)
	{attribute 'hide'}
	METHOD FB_init : BOOL
	VAR_INPUT
		(*  if TRUE, the retain variables are initialized (warm start / cold start) *)
		bInitRetains : BOOL;
		(*  if TRUE, the instance afterwards gets moved into the copy code (online change) *)
		bInCopyCode : BOOL;
	END_VAR
END_METHOD


	(* Internal method *)
	{attribute 'hide'}
	METHOD FB_exit : BOOL
	VAR_INPUT
		(*  if TRUE, the exit method is called for exiting an instance that is copied afterwards (online change). *)
		bInCopyCode : BOOL;
	END_VAR
END_METHOD


	(* Append a smooth transition from the current end of the path
				    to the specified position. *)
	METHOD AppendPosition
	VAR_IN_OUT
		(* The position to append. *)
 {attribute 'GUID' := '79961EF3-A89D-96D9-D6D0-3818573828BC'}
				position : PositionXYC;
	END_VAR
END_METHOD


	(* Append a smooth transition from the current end of the path
				    to the specified position. *)
	METHOD AppendPositionXYC
	VAR_INPUT
		(* x-component of the position to append. *)
		x : LREAL;
		(* y-component of the position to append. *)
		y : LREAL;
		(* c-component of the position to append in degrees [Â°]. *)
		c : LREAL;
	END_VAR
END_METHOD


	(* Append a line to this path. *)
	METHOD AppendLine
	VAR_IN_OUT
		(* Start position of the line. *)
 {attribute 'GUID' := '79961EF3-A89D-96D9-D6D0-3818573828BC'}
				startPos : PositionXYC;
		(* End position of the line. *)
 {attribute 'GUID' := '79961EF3-A89D-96D9-D6D0-3818573828BC'}
				endPos : PositionXYC;
	END_VAR
END_METHOD


	(* Append a circle to this path. *)
	METHOD AppendCircle
	VAR_IN_OUT
		(* Start position of the circle. *)
 {attribute 'GUID' := '79961EF3-A89D-96D9-D6D0-3818573828BC'}
				startPos : PositionXYC;
		(* End position of the circle. *)
 {attribute 'GUID' := '79961EF3-A89D-96D9-D6D0-3818573828BC'}
				endPos : PositionXYC;
		(* Center of the circle. *)
 {attribute 'GUID' := 'FCACA74E-C57F-9E9F-C3FF-7BECD9A9CD0E'}
				center : PositionXY;
	END_VAR
	VAR_INPUT
		(* Set whether the circle runs clockwise or counter-clockwise. *)
		clockwise : BOOL;
	END_VAR
END_METHOD


	(* Appends a smooth transition from the end of this path
				      to the start of the other path, locking further changes of this path. *)
	METHOD EndAtPath
	VAR_IN_OUT
		(* The other path. *)
 {attribute 'GUID' := '6E12F92E-6BF9-9AF0-D560-BBDFBB18383E'}
				path : PathXYC;
	END_VAR
END_METHOD


	(* Appends a smooth transition from the start of this path
				      to the end of the other path, locking further changes of the other path. *)
	METHOD StartFromPath
	VAR_IN_OUT
		(* The other path. *)
 {attribute 'GUID' := '6E12F92E-6BF9-9AF0-D560-BBDFBB18383E'}
				path : PathXYC;
	END_VAR
END_METHOD


	(* Connect start and end position.
				      A smooth transition is added as long as start and end positin are not identical.
				      This operation finalizes this path definition and locks it against further modifications. *)
	METHOD CloseLoop
END_METHOD


	(* Empty all current path definitions and reset the path back to an empty state. *)
	METHOD Clear
END_METHOD


	(* Get the start position of the path. *)
	METHOD GetStartPosition
	VAR_IN_OUT
		(* The current start position of the path. *)
 {attribute 'GUID' := '79961EF3-A89D-96D9-D6D0-3818573828BC'}
				startPosition : PositionXYC;
	END_VAR
END_METHOD


	(* Get the end position of the segment. *)
	METHOD GetEndPosition
	VAR_IN_OUT
		(* The current end position of the segment. *)
 {attribute 'GUID' := '79961EF3-A89D-96D9-D6D0-3818573828BC'}
				endPosition : PositionXYC;
	END_VAR
END_METHOD


	(* Get a position on the path at a specific arclength value. *)
	METHOD GetPositionAt
	VAR_INPUT
		(* Arc length value where the position is evaluated. *)
		arcLength : LREAL;
	END_VAR
	VAR_IN_OUT
		(* The position at the specified arc parameter. *)
 {attribute 'GUID' := '79961EF3-A89D-96D9-D6D0-3818573828BC'}
				position : PositionXYC;
	END_VAR
END_METHOD


	(* Get the dynamic information when moving along a path
				    with specific arclength value and dynamic changes. *)
	METHOD GetStateAt
	VAR_INPUT
		(* Arc length value where the position is evaluated. *)
		arcLength : LREAL;
		(* Velocity of the arc length parameter. *)
		arcVelocity : LREAL;
		(* Acceleration of the arc length parameter. *)
		arcAcceleration : LREAL;
	END_VAR
	VAR_IN_OUT
		(* The position at the specified arc parameter. *)
 {attribute 'GUID' := '79961EF3-A89D-96D9-D6D0-3818573828BC'}
				position : PositionXYC;
		(* The velocity at the specified dynamic state. *)
 {attribute 'GUID' := 'CD4C5ADD-3316-9B2E-DDE7-F563BE7C8FB2'}
				velocity : TangentXYC;
		(* The acceleration at the specified dynamic state. *)
 {attribute 'GUID' := 'CD4C5ADD-3316-9B2E-DDE7-F563BE7C8FB2'}
				acceleration : TangentXYC;
	END_VAR
END_METHOD

END_FUNCTION_BLOCK

// POUs/Shapes/Geometry3D/Container3D

	{attribute 'c++_compatible'}
	{attribute 'external_name' := 'Container3D_GUID_FA0F9463_565F_93EC_EB62_A449A3F269C0'}
	{attribute 'TcIecLibraryType'}
	{attribute 'no_explicit_call' :='do not call this POU directly'}
	{attribute 'no_assign'}
	FUNCTION_BLOCK Container3D EXTENDS Geometry3D


	(* Internal method *)
	METHOD FB_init : BOOL
	VAR_INPUT
		(*  if TRUE, the retain variables are initialized (warm start / cold start) *)
		bInitRetains : BOOL;
		(*  if TRUE, the instance afterwards gets moved into the copy code (online change) *)
		bInCopyCode : BOOL;
	END_VAR
END_METHOD


	(* Internal method *)
	{attribute 'hide'}
	METHOD FB_exit : BOOL
	VAR_INPUT
		(*  if TRUE, the exit method is called for exiting an instance that is copied afterwards (online change). *)
		bInCopyCode : BOOL;
	END_VAR
END_METHOD


	(* Add a geometry to the container. *)
	METHOD AddElement : UDINT
	VAR_IN_OUT
		(* The geometry to add. *)
 {attribute 'GUID' := '7BE2BD76-5981-9401-DE5E-712E37B15AA0'}
				geometry : Geometry3D;
	END_VAR
END_METHOD


	(* Remove a specified geometry from the container. *)
	METHOD RemoveElement
	VAR_INPUT
		(* Identifier of the geometry to remove. *)
		id : UDINT;
	END_VAR
END_METHOD


	(* Remove all geometries from container. *)
	METHOD Clear
END_METHOD


	(* Get the number of geometry elements in container. *)
	METHOD GetCount : UDINT
END_METHOD

END_FUNCTION_BLOCK

// POUs/Shapes/Geometry3D/Extrude3D

	{attribute 'c++_compatible'}
	{attribute 'external_name' := 'Extrude3D_GUID_B0F7556C_9699_90A0_EF34_9D8E02AEEB5B'}
	{attribute 'TcIecLibraryType'}
	{attribute 'no_explicit_call' :='do not call this POU directly'}
	{attribute 'no_assign'}
	FUNCTION_BLOCK Extrude3D EXTENDS Geometry3D


	(* Internal method *)
	METHOD FB_init : BOOL
	VAR_INPUT
		(*  if TRUE, the retain variables are initialized (warm start / cold start) *)
		bInitRetains : BOOL;
		(*  if TRUE, the instance afterwards gets moved into the copy code (online change) *)
		bInCopyCode : BOOL;
	END_VAR
END_METHOD


	(* Internal method *)
	{attribute 'hide'}
	METHOD FB_exit : BOOL
	VAR_INPUT
		(*  if TRUE, the exit method is called for exiting an instance that is copied afterwards (online change). *)
		bInCopyCode : BOOL;
	END_VAR
END_METHOD


	(* Define the extrude geometry with a path and a array of xy-points *)
	METHOD DefineByPath : BOOL
	VAR_IN_OUT
		(* Cross section values *)
 {attribute 'GUID' := 'FCACA74E-C57F-9E9F-C3FF-7BECD9A9CD0E'}
				PointerToCrossSection : POINTER TO PositionXY;
	END_VAR
	VAR_INPUT
		(* Number of cross section points *)
		NumberOfCrossSectionPoints : UDINT;
	END_VAR
	VAR_IN_OUT
		(* The path *)
 {attribute 'GUID' := '481DB202-0307-9E42-E144-16928531132C'}
				Path : PathXYZ;
	END_VAR
	VAR_INPUT
		(* Number of path points *)
		NumberOfPathPoints : UDINT;
	END_VAR
END_METHOD

END_FUNCTION_BLOCK

// POUs/Paths/Components/PathXYZ

	{attribute 'c++_compatible'}
	{attribute 'external_name' := 'PathXYZ_GUID_481DB202_0307_9E42_E144_16928531132C'}
	{attribute 'TcIecLibraryType'}
	{attribute 'no_explicit_call' :='do not call this POU directly'}
	{attribute 'no_assign'}
	(* A path in the xy-plane with an additional orientation at every path position. *)
	FUNCTION_BLOCK PathXYZ EXTENDS IPlcPath3D


	(* Internal method *)
	{attribute 'hide'}
	METHOD FB_init : BOOL
	VAR_INPUT
		(*  if TRUE, the retain variables are initialized (warm start / cold start) *)
		bInitRetains : BOOL;
		(*  if TRUE, the instance afterwards gets moved into the copy code (online change) *)
		bInCopyCode : BOOL;
	END_VAR
END_METHOD


	(* Internal method *)
	{attribute 'hide'}
	METHOD FB_exit : BOOL
	VAR_INPUT
		(*  if TRUE, the exit method is called for exiting an instance that is copied afterwards (online change). *)
		bInCopyCode : BOOL;
	END_VAR
END_METHOD


	(* Append a smooth transition from the current end of the path
				    to the specified position. *)
	METHOD AppendPosition
	VAR_IN_OUT
		(* The position to append. *)
 {attribute 'GUID' := '40E6105C-AAE1-907F-E93C-27FE8D6C7544'}
				position : Position3D;
	END_VAR
END_METHOD


	(* Append a smooth transition from the current end of the path
				    to the specified position. *)
	METHOD AppendPositionXYZ
	VAR_INPUT
		(* x-component of the position to append. *)
		x : LREAL;
		(* y-component of the position to append. *)
		y : LREAL;
		(* z-component of the position to append. *)
		c : LREAL;
	END_VAR
END_METHOD


	(* Append a line to this path. *)
	METHOD AppendLine
	VAR_IN_OUT
		(* Start position of the line. *)
 {attribute 'GUID' := '40E6105C-AAE1-907F-E93C-27FE8D6C7544'}
				startPos : Position3D;
		(* End position of the line. *)
 {attribute 'GUID' := '40E6105C-AAE1-907F-E93C-27FE8D6C7544'}
				endPos : Position3D;
	END_VAR
END_METHOD


	(* Append a smooth transition from the current end of the path
				    to the specified position. *)
	METHOD AppendLineXYZ
	VAR_INPUT
		(* x-component of the start position. *)
		x0 : LREAL;
		(* y-component of the start position. *)
		y0 : LREAL;
		(* z-component of the start position. *)
		z0 : LREAL;
		(* x-component of the end position. *)
		x1 : LREAL;
		(* y-component of the end position. *)
		y1 : LREAL;
		(* z-component of the end position. *)
		z1 : LREAL;
	END_VAR
END_METHOD


	(* Append a circle to this path. *)
	METHOD AppendCircle
	VAR_IN_OUT
		(* Start position of the circle. *)
 {attribute 'GUID' := '40E6105C-AAE1-907F-E93C-27FE8D6C7544'}
				startPos : Position3D;
		(* End position of the circle. *)
 {attribute 'GUID' := '40E6105C-AAE1-907F-E93C-27FE8D6C7544'}
				endPos : Position3D;
		(* Center of the circle. *)
 {attribute 'GUID' := 'FCACA74E-C57F-9E9F-C3FF-7BECD9A9CD0E'}
				center : PositionXY;
	END_VAR
	VAR_INPUT
		(* Set whether the circle runs clockwise or counter-clockwise. *)
		clockwise : BOOL;
	END_VAR
END_METHOD


	(* Append a smooth transition from the current end of the path
				    to the specified position with tangent. *)
	METHOD AppendPositionTangent
	VAR_IN_OUT
		(* The position to append. *)
 {attribute 'GUID' := '40E6105C-AAE1-907F-E93C-27FE8D6C7544'}
				position : Position3D;
		(* The tangent to append *)
 {attribute 'GUID' := '9F987066-55C3-9A71-FEA1-9CB49A451CD6'}
				tangent : Tangent3D;
	END_VAR
END_METHOD


	(* Get the start position of the path. *)
	METHOD GetStartPosition
	VAR_IN_OUT
		(* The current start position of the path. *)
 {attribute 'GUID' := '40E6105C-AAE1-907F-E93C-27FE8D6C7544'}
				startPosition : Position3D;
	END_VAR
END_METHOD


	(* Get the end position of the segment. *)
	METHOD GetEndPosition
	VAR_IN_OUT
		(* The current end position of the segment. *)
 {attribute 'GUID' := '40E6105C-AAE1-907F-E93C-27FE8D6C7544'}
				endPosition : Position3D;
	END_VAR
END_METHOD


	(* Get a position on the path at a specific arclength value. *)
	METHOD GetPositionAt
	VAR_INPUT
		(* Arc length value where the position is evaluated. *)
		arcLength : LREAL;
	END_VAR
	VAR_IN_OUT
		(* The position at the specified arc parameter. *)
 {attribute 'GUID' := '40E6105C-AAE1-907F-E93C-27FE8D6C7544'}
				position : Position3D;
	END_VAR
END_METHOD


	(* Get the dynamic information when moving along a path
				    with specific arclength value and dynamic changes. *)
	METHOD GetStateAt
	VAR_INPUT
		(* Arc length value where the position is evaluated. *)
		arcLength : LREAL;
		(* Velocity of the arc length parameter. *)
		arcVelocity : LREAL;
		(* Acceleration of the arc length parameter. *)
		arcAcceleration : LREAL;
	END_VAR
	VAR_IN_OUT
		(* The position at the specified arc parameter. *)
 {attribute 'GUID' := '40E6105C-AAE1-907F-E93C-27FE8D6C7544'}
				position : Position3D;
		(* The velocity at the specified dynamic state. *)
 {attribute 'GUID' := '9F987066-55C3-9A71-FEA1-9CB49A451CD6'}
				velocity : Tangent3D;
		(* The acceleration at the specified dynamic state. *)
 {attribute 'GUID' := '9F987066-55C3-9A71-FEA1-9CB49A451CD6'}
				acceleration : Tangent3D;
	END_VAR
END_METHOD

END_FUNCTION_BLOCK

// POUs/Paths/Components/PathXY

	{attribute 'c++_compatible'}
	{attribute 'external_name' := 'PathXY_GUID_AFFA2879_6880_90AC_CE5A_A46DB9773315'}
	{attribute 'TcIecLibraryType'}
	{attribute 'no_explicit_call' :='do not call this POU directly'}
	{attribute 'no_assign'}
	(* A path in the xy-plane. *)
	FUNCTION_BLOCK PathXY EXTENDS IPlcPath2D


	(* Internal method *)
	{attribute 'hide'}
	METHOD FB_init : BOOL
	VAR_INPUT
		(*  if TRUE, the retain variables are initialized (warm start / cold start) *)
		bInitRetains : BOOL;
		(*  if TRUE, the instance afterwards gets moved into the copy code (online change) *)
		bInCopyCode : BOOL;
	END_VAR
END_METHOD


	(* Internal method *)
	{attribute 'hide'}
	METHOD FB_exit : BOOL
	VAR_INPUT
		(*  if TRUE, the exit method is called for exiting an instance that is copied afterwards (online change). *)
		bInCopyCode : BOOL;
	END_VAR
END_METHOD


	(* Append a smooth transition from the current end of the path
				    to the specified position. *)
	METHOD AppendPosition
	VAR_IN_OUT
		(* The position to append. *)
 {attribute 'GUID' := 'FCACA74E-C57F-9E9F-C3FF-7BECD9A9CD0E'}
				position : PositionXY;
	END_VAR
END_METHOD


	(* Append a smooth transition from the current end of the path
				    to the specified position. *)
	METHOD AppendPositionXY
	VAR_INPUT
		(* x-component of the position to append. *)
		x : LREAL;
		(* y-component of the position to append. *)
		y : LREAL;
	END_VAR
END_METHOD


	(* Append a line to this path. *)
	METHOD AppendLine
	VAR_IN_OUT
		(* Start position of the line. *)
 {attribute 'GUID' := 'FCACA74E-C57F-9E9F-C3FF-7BECD9A9CD0E'}
				startPos : PositionXY;
		(* End position of the line. *)
 {attribute 'GUID' := 'FCACA74E-C57F-9E9F-C3FF-7BECD9A9CD0E'}
				endPos : PositionXY;
	END_VAR
END_METHOD


	(* Append a circle to this path. *)
	METHOD AppendCircle
	VAR_IN_OUT
		(* Start position of the circle. *)
 {attribute 'GUID' := 'FCACA74E-C57F-9E9F-C3FF-7BECD9A9CD0E'}
				startPos : PositionXY;
		(* End position of the circle. *)
 {attribute 'GUID' := 'FCACA74E-C57F-9E9F-C3FF-7BECD9A9CD0E'}
				endPos : PositionXY;
		(* Center of the circle. *)
 {attribute 'GUID' := 'FCACA74E-C57F-9E9F-C3FF-7BECD9A9CD0E'}
				center : PositionXY;
	END_VAR
	VAR_INPUT
		(* Set whether the circle runs clockwise or counter-clockwise. *)
		clockwise : BOOL;
	END_VAR
END_METHOD


	(* Get the start position of the path. *)
	METHOD GetStartPosition
	VAR_IN_OUT
		(* The current start position of the path. *)
 {attribute 'GUID' := 'FCACA74E-C57F-9E9F-C3FF-7BECD9A9CD0E'}
				startPosition : PositionXY;
	END_VAR
END_METHOD


	(* Get the end position of the segment. *)
	METHOD GetEndPosition
	VAR_IN_OUT
		(* The current end position of the segment. *)
 {attribute 'GUID' := 'FCACA74E-C57F-9E9F-C3FF-7BECD9A9CD0E'}
				endPosition : PositionXY;
	END_VAR
END_METHOD


	(* Get a position on the path at a specific arclength value. *)
	METHOD GetPositionAt
	VAR_INPUT
		(* Arc length value where the position is evaluated. *)
		arcLength : LREAL;
	END_VAR
	VAR_IN_OUT
		(* The position at the specified arc parameter. *)
 {attribute 'GUID' := 'FCACA74E-C57F-9E9F-C3FF-7BECD9A9CD0E'}
				position : PositionXY;
	END_VAR
END_METHOD


	(* Get the dynamic information when moving along a path
				    with specific arclength value and dynamic changes. *)
	METHOD GetStateAt
	VAR_INPUT
		(* Arc length value where the position is evaluated. *)
		arcLength : LREAL;
		(* Velocity of the arc length parameter. *)
		arcVelocity : LREAL;
		(* Acceleration of the arc length parameter. *)
		arcAcceleration : LREAL;
	END_VAR
	VAR_IN_OUT
		(* The position at the specified arc parameter. *)
 {attribute 'GUID' := 'FCACA74E-C57F-9E9F-C3FF-7BECD9A9CD0E'}
				position : PositionXY;
		(* The velocity at the specified dynamic state. *)
 {attribute 'GUID' := '4CE6AEBB-A122-94B9-C485-29D927BD5C71'}
				velocity : TangentXY;
		(* The acceleration at the specified dynamic state. *)
 {attribute 'GUID' := '4CE6AEBB-A122-94B9-C485-29D927BD5C71'}
				acceleration : TangentXY;
	END_VAR
END_METHOD

END_FUNCTION_BLOCK

// POUs/Shapes/Geometry2D/1D/Line2D

	{attribute 'c++_compatible'}
	{attribute 'external_name' := 'Line2D_GUID_BB734A6A_B90B_9815_C25D_D5A4B1FD5737'}
	{attribute 'TcIecLibraryType'}
	{attribute 'no_explicit_call' :='do not call this POU directly'}
	{attribute 'no_assign'}
	(* 2D Geometry Line *)
	FUNCTION_BLOCK Line2D EXTENDS Geometry2D


	(* Internal method *)
	METHOD FB_init : BOOL
	VAR_INPUT
		(*  if TRUE, the retain variables are initialized (warm start / cold start) *)
		bInitRetains : BOOL;
		(*  if TRUE, the instance afterwards gets moved into the copy code (online change) *)
		bInCopyCode : BOOL;
	END_VAR
END_METHOD


	(* Internal method *)
	{attribute 'hide'}
	METHOD FB_exit : BOOL
	VAR_INPUT
		(*  if TRUE, the exit method is called for exiting an instance that is copied afterwards (online change). *)
		bInCopyCode : BOOL;
	END_VAR
END_METHOD


	(* Define a line by two positions. *)
	METHOD DefineByPositions
	VAR_IN_OUT
		(* 1st position on the line to define. *)
 {attribute 'GUID' := 'FCACA74E-C57F-9E9F-C3FF-7BECD9A9CD0E'}
				position0 : PositionXY;
		(* 2nd position on the line to define. *)
 {attribute 'GUID' := 'FCACA74E-C57F-9E9F-C3FF-7BECD9A9CD0E'}
				position1 : PositionXY;
	END_VAR
END_METHOD


	(* Define a line by a position on the line and its direction. *)
	METHOD DefineByDirection
	VAR_IN_OUT
		(* Position on the line *)
 {attribute 'GUID' := 'FCACA74E-C57F-9E9F-C3FF-7BECD9A9CD0E'}
				position : PositionXY;
		(* Direction of the line *)
 {attribute 'GUID' := '4CE6AEBB-A122-94B9-C485-29D927BD5C71'}
				direction : TangentXY;
	END_VAR
END_METHOD


	(* Set the direction of the line. *)
	METHOD SetDirection
	VAR_IN_OUT
		(* The direction to set. *)
 {attribute 'GUID' := '4CE6AEBB-A122-94B9-C485-29D927BD5C71'}
				direction : TangentXY;
	END_VAR
END_METHOD


	(* Get the direction of the line. *)
	METHOD GetDirection
	VAR_IN_OUT
		(* The current direction of the line. *)
 {attribute 'GUID' := '4CE6AEBB-A122-94B9-C485-29D927BD5C71'}
				direction : TangentXY;
	END_VAR
END_METHOD


	(* Get a position on the line at a specific arclength value. *)
	METHOD GetPositionAt
	VAR_INPUT
		(* Arc length value where the position is evaluated. *)
		arcLength : LREAL;
	END_VAR
	VAR_IN_OUT
		(* The position at the specified arc parameter. *)
 {attribute 'GUID' := '79961EF3-A89D-96D9-D6D0-3818573828BC'}
				position : PositionXYC;
	END_VAR
END_METHOD

END_FUNCTION_BLOCK

// POUs/Shapes/Geometry2D/1D/Segment2D

	{attribute 'c++_compatible'}
	{attribute 'external_name' := 'Segment2D_GUID_DA82AA6F_B88D_900B_C10B_A07419B1C4ED'}
	{attribute 'TcIecLibraryType'}
	{attribute 'no_explicit_call' :='do not call this POU directly'}
	{attribute 'no_assign'}
	FUNCTION_BLOCK Segment2D EXTENDS Geometry2D


	(* Internal method *)
	METHOD FB_init : BOOL
	VAR_INPUT
		(*  if TRUE, the retain variables are initialized (warm start / cold start) *)
		bInitRetains : BOOL;
		(*  if TRUE, the instance afterwards gets moved into the copy code (online change) *)
		bInCopyCode : BOOL;
	END_VAR
END_METHOD


	(* Internal method *)
	{attribute 'hide'}
	METHOD FB_exit : BOOL
	VAR_INPUT
		(*  if TRUE, the exit method is called for exiting an instance that is copied afterwards (online change). *)
		bInCopyCode : BOOL;
	END_VAR
END_METHOD


	(* Set the start position of the segment. *)
	METHOD SetStartPosition
	VAR_IN_OUT
		(* Start position of the segment to set. *)
 {attribute 'GUID' := 'FCACA74E-C57F-9E9F-C3FF-7BECD9A9CD0E'}
				startPos : PositionXY;
	END_VAR
END_METHOD


	(* Set the start position of the segment. *)
	METHOD SetStartPositionXY
	VAR_INPUT
		(* x-component of the start position. *)
		x : LREAL;
		(* y-component of the start position. *)
		y : LREAL;
	END_VAR
END_METHOD


	(* Set the end position of the segment. *)
	METHOD SetEndPosition
	VAR_IN_OUT
		(* End position of the segment to set. *)
 {attribute 'GUID' := 'FCACA74E-C57F-9E9F-C3FF-7BECD9A9CD0E'}
				endPos : PositionXY;
	END_VAR
END_METHOD


	(* Set the end position of the segment. *)
	METHOD SetEndPositionXY
	VAR_INPUT
		(* x-component of the end position. *)
		x : LREAL;
		(* y-component of the end position. *)
		y : LREAL;
	END_VAR
END_METHOD


	(* Get the x-component of the segment length in respect to the root coordinate system. *)
	METHOD Get_dX : LREAL
END_METHOD


	(* Get the y-component of the segment length in respect to the root coordinate system. *)
	METHOD Get_dY : LREAL
END_METHOD


	(* Get the length of the segment. *)
	METHOD GetLength : LREAL
END_METHOD


	(* Get the start position of the segment. *)
	METHOD GetStartPosition
	VAR_IN_OUT
		(* The current start position of the segment. *)
 {attribute 'GUID' := 'FCACA74E-C57F-9E9F-C3FF-7BECD9A9CD0E'}
				startPosition : PositionXY;
	END_VAR
END_METHOD


	(* Get the end position of the segment. *)
	METHOD GetEndPosition
	VAR_IN_OUT
		(* The current end position of the segment. *)
 {attribute 'GUID' := 'FCACA74E-C57F-9E9F-C3FF-7BECD9A9CD0E'}
				endPosition : PositionXY;
	END_VAR
END_METHOD


	(* Get the direction of the segment. *)
	METHOD GetDirection
	VAR_IN_OUT
		(* The current direction of the segment. *)
 {attribute 'GUID' := '4CE6AEBB-A122-94B9-C485-29D927BD5C71'}
				direction : TangentXY;
	END_VAR
END_METHOD


	(* Get a position on the segment at a specific arclength value. *)
	METHOD GetPositionAt
	VAR_INPUT
		(* Arc length value where the position is evaluated. *)
		arcLength : LREAL;
	END_VAR
	VAR_IN_OUT
		(* The position at the specified arc parameter. *)
 {attribute 'GUID' := '79961EF3-A89D-96D9-D6D0-3818573828BC'}
				position : PositionXYC;
	END_VAR
END_METHOD

END_FUNCTION_BLOCK

// POUs/Shapes/Geometry2D/1D/Circle2D

	{attribute 'c++_compatible'}
	{attribute 'external_name' := 'Circle2D_GUID_8DC5791C_B411_93C2_F3D1_82443F18814C'}
	{attribute 'TcIecLibraryType'}
	{attribute 'no_explicit_call' :='do not call this POU directly'}
	{attribute 'no_assign'}
	FUNCTION_BLOCK Circle2D EXTENDS Geometry2D


	(* Internal method *)
	METHOD FB_init : BOOL
	VAR_INPUT
		(*  if TRUE, the retain variables are initialized (warm start / cold start) *)
		bInitRetains : BOOL;
		(*  if TRUE, the instance afterwards gets moved into the copy code (online change) *)
		bInCopyCode : BOOL;
	END_VAR
END_METHOD


	(* Internal method *)
	{attribute 'hide'}
	METHOD FB_exit : BOOL
	VAR_INPUT
		(*  if TRUE, the exit method is called for exiting an instance that is copied afterwards (online change). *)
		bInCopyCode : BOOL;
	END_VAR
END_METHOD


	(* Get the length of the circle. *)
	METHOD GetLength : LREAL
END_METHOD


	(* Get a position on the circle at a specific arclength value. *)
	METHOD GetPositionAt
	VAR_INPUT
		(* Arc length value where the position is evaluated. *)
		arcLength : LREAL;
	END_VAR
	VAR_IN_OUT
		(* The position at the specified arc parameter. *)
 {attribute 'GUID' := '79961EF3-A89D-96D9-D6D0-3818573828BC'}
				position : PositionXYC;
	END_VAR
END_METHOD


	PROPERTY radius : LREAL
GET
END_GET
SET
END_SET
END_PROPERTY

END_FUNCTION_BLOCK

// POUs/Shapes/Geometry2D/2D/Disc2D

	{attribute 'c++_compatible'}
	{attribute 'external_name' := 'Disc2D_GUID_703205F2_2ACA_9A34_EB93_09253B098460'}
	{attribute 'TcIecLibraryType'}
	{attribute 'no_explicit_call' :='do not call this POU directly'}
	{attribute 'no_assign'}
	FUNCTION_BLOCK Disc2D EXTENDS Geometry2D


	(* Internal method *)
	METHOD FB_init : BOOL
	VAR_INPUT
		(*  if TRUE, the retain variables are initialized (warm start / cold start) *)
		bInitRetains : BOOL;
		(*  if TRUE, the instance afterwards gets moved into the copy code (online change) *)
		bInCopyCode : BOOL;
	END_VAR
END_METHOD


	(* Internal method *)
	{attribute 'hide'}
	METHOD FB_exit : BOOL
	VAR_INPUT
		(*  if TRUE, the exit method is called for exiting an instance that is copied afterwards (online change). *)
		bInCopyCode : BOOL;
	END_VAR
END_METHOD


	(* Get the area of the disc. *)
	METHOD GetArea : LREAL
END_METHOD


	PROPERTY radius : LREAL
GET
END_GET
SET
END_SET
END_PROPERTY

END_FUNCTION_BLOCK

// POUs/Shapes/Geometry2D/2D/Rectangle2D

	{attribute 'c++_compatible'}
	{attribute 'external_name' := 'Rectangle2D_GUID_5E10366F_AEAF_967C_F04B_B22C26EEAB72'}
	{attribute 'TcIecLibraryType'}
	{attribute 'no_explicit_call' :='do not call this POU directly'}
	{attribute 'no_assign'}
	FUNCTION_BLOCK Rectangle2D EXTENDS Geometry2D


	(* Internal method *)
	METHOD FB_init : BOOL
	VAR_INPUT
		(*  if TRUE, the retain variables are initialized (warm start / cold start) *)
		bInitRetains : BOOL;
		(*  if TRUE, the instance afterwards gets moved into the copy code (online change) *)
		bInCopyCode : BOOL;
	END_VAR
END_METHOD


	(* Internal method *)
	{attribute 'hide'}
	METHOD FB_exit : BOOL
	VAR_INPUT
		(*  if TRUE, the exit method is called for exiting an instance that is copied afterwards (online change). *)
		bInCopyCode : BOOL;
	END_VAR
END_METHOD


	(* Set the dimensions of the rectangle. *)
	METHOD SetDimensions
	VAR_INPUT
		(* The width of the rectangle to set. *)
		width : LREAL;
		(* The height of the rectangle to set. *)
		height : LREAL;
	END_VAR
END_METHOD


	(* Get the area of the rectangle. *)
	METHOD GetArea : LREAL
END_METHOD


	PROPERTY width : LREAL
GET
END_GET
SET
END_SET
END_PROPERTY


	PROPERTY height : LREAL
GET
END_GET
SET
END_SET
END_PROPERTY

END_FUNCTION_BLOCK

// POUs/Shapes/Geometry2D/Functions/CheckCollision2D

	{attribute 'TcIecLibraryType'}
	{attribute 'external_name' := 'CheckCollision2D_GUID_E0A3A9E8_3456_9D82_FD09_2A14A2B19BF6'}
	(* Check if two geometries are currently colliding. *)
	FUNCTION CheckCollision2D : BOOL
	VAR_IN_OUT
		geometry0	:	IPlcGeometry2D;	(* 1st input geometry to check for collision. *)
		geometry1	:	IPlcGeometry2D;	(* 2nd input geometry to check of collision. *)
	END_VAR

END_FUNCTION

// POUs/Shapes/Geometry2D/Functions/GetDistance2D

	{attribute 'TcIecLibraryType'}
	{attribute 'external_name' := 'GetDistance2D_GUID_DF6CD210_F52D_9717_C945_2435170A466A'}
	(* Get the distance between two geometries. *)
	FUNCTION GetDistance2D : LREAL
	VAR_IN_OUT
		geometry0	:	IPlcGeometry2D;	(* 1st input geometry to calculate the distance of. *)
		geometry1	:	IPlcGeometry2D;	(* 2nd input geometry to calculate the distance of. *)
	END_VAR

END_FUNCTION

// POUs/Shapes/Geometry2D/Functions/GetLinkingLine2D

	{attribute 'TcIecLibraryType'}
	{attribute 'external_name' := 'GetLinkingLine2D_GUID_9987D22F_87DB_997A_ED3B_4BAE5E26E93C'}
	(* Get the shortest path between two geometries. *)
	FUNCTION GetLinkingLine2D : BOOL
	VAR_IN_OUT
		geometry0	:	IPlcGeometry2D;	(* 1st input geometry to calculate the linking line for. *)
		geometry1	:	IPlcGeometry2D;	(* 2nd input geometry to calculate the linking line for. *)
		linkingLine	:	Segment2D;	(* Return the resulting linking line. *)
	END_VAR

END_FUNCTION

// POUs/Shapes/Geometry3D/1D/Line3D

	{attribute 'c++_compatible'}
	{attribute 'external_name' := 'Line3D_GUID_B6CD31E5_EBFE_90E9_EBC4_B024E56B4F2C'}
	{attribute 'TcIecLibraryType'}
	{attribute 'no_explicit_call' :='do not call this POU directly'}
	{attribute 'no_assign'}
	(* 3D Geometry Line *)
	FUNCTION_BLOCK Line3D EXTENDS Geometry3D


	(* Internal method *)
	METHOD FB_init : BOOL
	VAR_INPUT
		(*  if TRUE, the retain variables are initialized (warm start / cold start) *)
		bInitRetains : BOOL;
		(*  if TRUE, the instance afterwards gets moved into the copy code (online change) *)
		bInCopyCode : BOOL;
	END_VAR
END_METHOD


	(* Internal method *)
	{attribute 'hide'}
	METHOD FB_exit : BOOL
	VAR_INPUT
		(*  if TRUE, the exit method is called for exiting an instance that is copied afterwards (online change). *)
		bInCopyCode : BOOL;
	END_VAR
END_METHOD


	(* Define a line by two positions. *)
	METHOD DefineByPositions
	VAR_IN_OUT
		(* 1st position on the line to define. *)
 {attribute 'GUID' := '40E6105C-AAE1-907F-E93C-27FE8D6C7544'}
				position0 : Position3D;
		(* 2nd position on the line to define. *)
 {attribute 'GUID' := '40E6105C-AAE1-907F-E93C-27FE8D6C7544'}
				position1 : Position3D;
	END_VAR
END_METHOD


	(* Define a line by a position on the line and its direction. *)
	METHOD DefineByDirection
	VAR_IN_OUT
		(* Position on the line. *)
 {attribute 'GUID' := '40E6105C-AAE1-907F-E93C-27FE8D6C7544'}
				position : Position3D;
		(* Direction of the line. *)
 {attribute 'GUID' := '9F987066-55C3-9A71-FEA1-9CB49A451CD6'}
				direction : Tangent3D;
	END_VAR
END_METHOD


	(* Set the direction of the line. *)
	METHOD SetDirection
	VAR_IN_OUT
		(* The direction to set. *)
 {attribute 'GUID' := '9F987066-55C3-9A71-FEA1-9CB49A451CD6'}
				direction : Tangent3D;
	END_VAR
END_METHOD


	(* Get the direction of the line. *)
	METHOD GetDirection
	VAR_IN_OUT
		(* The current direction of the line. *)
 {attribute 'GUID' := '9F987066-55C3-9A71-FEA1-9CB49A451CD6'}
				direction : Tangent3D;
	END_VAR
END_METHOD


	(* Get a position on the line at a specific arclength value. *)
	METHOD GetPositionAt
	VAR_INPUT
		(* Arc length value where the position is evaluated. *)
		arcLength : LREAL;
	END_VAR
	VAR_IN_OUT
		(* The position at the specified arc parameter. *)
 {attribute 'GUID' := '608A620D-3BBF-9A33-F5CB-39FFBA2AADD1'}
				position : PositionSE3;
	END_VAR
END_METHOD

END_FUNCTION_BLOCK

// POUs/Shapes/Geometry3D/1D/Segment3D

	{attribute 'c++_compatible'}
	{attribute 'external_name' := 'Segment3D_GUID_8B1C2377_5402_97CD_F3ED_CF9002FB8F7C'}
	{attribute 'TcIecLibraryType'}
	{attribute 'no_explicit_call' :='do not call this POU directly'}
	{attribute 'no_assign'}
	FUNCTION_BLOCK Segment3D EXTENDS Geometry3D


	(* Internal method *)
	METHOD FB_init : BOOL
	VAR_INPUT
		(*  if TRUE, the retain variables are initialized (warm start / cold start) *)
		bInitRetains : BOOL;
		(*  if TRUE, the instance afterwards gets moved into the copy code (online change) *)
		bInCopyCode : BOOL;
	END_VAR
END_METHOD


	(* Internal method *)
	{attribute 'hide'}
	METHOD FB_exit : BOOL
	VAR_INPUT
		(*  if TRUE, the exit method is called for exiting an instance that is copied afterwards (online change). *)
		bInCopyCode : BOOL;
	END_VAR
END_METHOD


	(* Set the start position of the segment. *)
	METHOD SetStartPosition
	VAR_IN_OUT
		(* Start position of the segment to set. *)
 {attribute 'GUID' := '40E6105C-AAE1-907F-E93C-27FE8D6C7544'}
				startPos : Position3D;
	END_VAR
END_METHOD


	(* Set the start position of the segment. *)
	METHOD SetStartPositionXYZ
	VAR_INPUT
		(* x-component of the start position. *)
		x : LREAL;
		(* y-component of the start position. *)
		y : LREAL;
		(* z-component of the start position. *)
		z : LREAL;
	END_VAR
END_METHOD


	(* Set the end position of the segment. *)
	METHOD SetEndPosition
	VAR_IN_OUT
		(* End position of the segment to set. *)
 {attribute 'GUID' := '40E6105C-AAE1-907F-E93C-27FE8D6C7544'}
				endPos : Position3D;
	END_VAR
END_METHOD


	(* Set the end position of the segment. *)
	METHOD SetEndPositionXYZ
	VAR_INPUT
		(* x-component of the end position. *)
		x : LREAL;
		(* y-component of the end position. *)
		y : LREAL;
		(* z-component of the end position. *)
		z : LREAL;
	END_VAR
END_METHOD


	(* Get the x-component of the segment length in respect to the root coordinate system. *)
	METHOD Get_dX : LREAL
END_METHOD


	(* Get the y-component of the segment length in respect to the root coordinate system. *)
	METHOD Get_dY : LREAL
END_METHOD


	(* Get the z-component of the segment length in respect to the root coordinate system. *)
	METHOD Get_dZ : LREAL
END_METHOD


	(* Get the length of the segment. *)
	METHOD GetLength : LREAL
END_METHOD


	(* Get the start position of the segment. *)
	METHOD GetStartPosition
	VAR_IN_OUT
		(* The current start position of the segment. *)
 {attribute 'GUID' := '40E6105C-AAE1-907F-E93C-27FE8D6C7544'}
				startPosition : Position3D;
	END_VAR
END_METHOD


	(* Get the end position of the segment. *)
	METHOD GetEndPosition
	VAR_IN_OUT
		(* The current end position of the segment. *)
 {attribute 'GUID' := '40E6105C-AAE1-907F-E93C-27FE8D6C7544'}
				endPosition : Position3D;
	END_VAR
END_METHOD


	(* Get the direction of the segment. *)
	METHOD GetDirection
	VAR_IN_OUT
		(* The current direction of the segment. *)
 {attribute 'GUID' := '9F987066-55C3-9A71-FEA1-9CB49A451CD6'}
				direction : Tangent3D;
	END_VAR
END_METHOD


	(* Get a position on the segment at a specific arclength value. *)
	METHOD GetPositionAt
	VAR_INPUT
		(* Arc length value where the position is evaluated. *)
		arcLength : LREAL;
	END_VAR
	VAR_IN_OUT
		(* The position at the specified arc parameter. *)
 {attribute 'GUID' := '608A620D-3BBF-9A33-F5CB-39FFBA2AADD1'}
				position : PositionSE3;
	END_VAR
END_METHOD

END_FUNCTION_BLOCK

// POUs/Shapes/Geometry3D/1D/Circle3D

	{attribute 'c++_compatible'}
	{attribute 'external_name' := 'Circle3D_GUID_43AAFB90_68EC_9773_E754_5DAA37F23B11'}
	{attribute 'TcIecLibraryType'}
	{attribute 'no_explicit_call' :='do not call this POU directly'}
	{attribute 'no_assign'}
	FUNCTION_BLOCK Circle3D EXTENDS Geometry3D


	(* Internal method *)
	METHOD FB_init : BOOL
	VAR_INPUT
		(*  if TRUE, the retain variables are initialized (warm start / cold start) *)
		bInitRetains : BOOL;
		(*  if TRUE, the instance afterwards gets moved into the copy code (online change) *)
		bInCopyCode : BOOL;
	END_VAR
END_METHOD


	(* Internal method *)
	{attribute 'hide'}
	METHOD FB_exit : BOOL
	VAR_INPUT
		(*  if TRUE, the exit method is called for exiting an instance that is copied afterwards (online change). *)
		bInCopyCode : BOOL;
	END_VAR
END_METHOD


	(* Set the normal vector of the circle. *)
	METHOD SetNormal
	VAR_IN_OUT
		(* Normal vector to set. *)
 {attribute 'GUID' := '9F987066-55C3-9A71-FEA1-9CB49A451CD6'}
				normal : Tangent3D;
	END_VAR
END_METHOD


	(* Get the length of the circle. *)
	METHOD GetLength : LREAL
END_METHOD


	(* Get the normal vector of the circle. *)
	METHOD GetNormal
	VAR
		(* The current normal vector of the circle. *)
 {attribute 'GUID' := '9F987066-55C3-9A71-FEA1-9CB49A451CD6'}
				normal : Tangent3D;
	END_VAR
END_METHOD


	(* Get a position on the circle at a specific arclength value. *)
	METHOD GetPositionAt
	VAR_INPUT
		(* Arc length value where the position is evaluated. *)
		arcLength : LREAL;
	END_VAR
	VAR_IN_OUT
		(* The position at the specified arc parameter. *)
 {attribute 'GUID' := '608A620D-3BBF-9A33-F5CB-39FFBA2AADD1'}
				position : PositionSE3;
	END_VAR
END_METHOD


	PROPERTY radius : LREAL
GET
END_GET
SET
END_SET
END_PROPERTY

END_FUNCTION_BLOCK

// POUs/Shapes/Geometry3D/2D/Plane3D

	{attribute 'c++_compatible'}
	{attribute 'external_name' := 'Plane3D_GUID_B29A19E1_6161_9CA2_CC4A_05DA1A4D6E04'}
	{attribute 'TcIecLibraryType'}
	{attribute 'no_explicit_call' :='do not call this POU directly'}
	{attribute 'no_assign'}
	FUNCTION_BLOCK Plane3D EXTENDS Geometry3D


	(* Internal method *)
	METHOD FB_init : BOOL
	VAR_INPUT
		(*  if TRUE, the retain variables are initialized (warm start / cold start) *)
		bInitRetains : BOOL;
		(*  if TRUE, the instance afterwards gets moved into the copy code (online change) *)
		bInCopyCode : BOOL;
	END_VAR
END_METHOD


	(* Internal method *)
	{attribute 'hide'}
	METHOD FB_exit : BOOL
	VAR_INPUT
		(*  if TRUE, the exit method is called for exiting an instance that is copied afterwards (online change). *)
		bInCopyCode : BOOL;
	END_VAR
END_METHOD


	(* Set the normal of the plane. *)
	METHOD SetNormal
	VAR_IN_OUT
		(* The normal vector to set. *)
 {attribute 'GUID' := '9F987066-55C3-9A71-FEA1-9CB49A451CD6'}
				normal : Tangent3D;
	END_VAR
END_METHOD


	(* Get the normal vector of the plane. *)
	METHOD GetNormal
	VAR
		(* The current normal vector of the plane. *)
 {attribute 'GUID' := '9F987066-55C3-9A71-FEA1-9CB49A451CD6'}
				normal : Tangent3D;
	END_VAR
END_METHOD

END_FUNCTION_BLOCK

// POUs/Shapes/Geometry3D/2D/Disc3D

	{attribute 'c++_compatible'}
	{attribute 'external_name' := 'Disc3D_GUID_2824F73E_F382_90B6_C6E4_52687B4B0046'}
	{attribute 'TcIecLibraryType'}
	{attribute 'no_explicit_call' :='do not call this POU directly'}
	{attribute 'no_assign'}
	FUNCTION_BLOCK Disc3D EXTENDS Geometry3D


	(* Internal method *)
	METHOD FB_init : BOOL
	VAR_INPUT
		(*  if TRUE, the retain variables are initialized (warm start / cold start) *)
		bInitRetains : BOOL;
		(*  if TRUE, the instance afterwards gets moved into the copy code (online change) *)
		bInCopyCode : BOOL;
	END_VAR
END_METHOD


	(* Internal method *)
	{attribute 'hide'}
	METHOD FB_exit : BOOL
	VAR_INPUT
		(*  if TRUE, the exit method is called for exiting an instance that is copied afterwards (online change). *)
		bInCopyCode : BOOL;
	END_VAR
END_METHOD


	(* Set the normal vector of the disc. *)
	METHOD SetNormal
	VAR_IN_OUT
		(* The normal to set. *)
 {attribute 'GUID' := '9F987066-55C3-9A71-FEA1-9CB49A451CD6'}
				normal : Tangent3D;
	END_VAR
END_METHOD


	(* Get the normal vector of the disc. *)
	METHOD GetNormal
	VAR
		(* The current normal vector of the disc. *)
 {attribute 'GUID' := '9F987066-55C3-9A71-FEA1-9CB49A451CD6'}
				normal : Tangent3D;
	END_VAR
END_METHOD


	(* Get the area of the disc. *)
	METHOD GetArea : LREAL
END_METHOD


	PROPERTY radius : LREAL
GET
END_GET
SET
END_SET
END_PROPERTY

END_FUNCTION_BLOCK

// POUs/Shapes/Geometry3D/2D/Rectangle3D

	{attribute 'c++_compatible'}
	{attribute 'external_name' := 'Rectangle3D_GUID_7AAA6473_2104_9821_E4E2_FDDCB1CCA078'}
	{attribute 'TcIecLibraryType'}
	{attribute 'no_explicit_call' :='do not call this POU directly'}
	{attribute 'no_assign'}
	FUNCTION_BLOCK Rectangle3D EXTENDS Geometry3D


	(* Internal method *)
	METHOD FB_init : BOOL
	VAR_INPUT
		(*  if TRUE, the retain variables are initialized (warm start / cold start) *)
		bInitRetains : BOOL;
		(*  if TRUE, the instance afterwards gets moved into the copy code (online change) *)
		bInCopyCode : BOOL;
	END_VAR
END_METHOD


	(* Internal method *)
	{attribute 'hide'}
	METHOD FB_exit : BOOL
	VAR_INPUT
		(*  if TRUE, the exit method is called for exiting an instance that is copied afterwards (online change). *)
		bInCopyCode : BOOL;
	END_VAR
END_METHOD


	(* Set the dimensions of the rectangle. *)
	METHOD SetDimensions
	VAR_INPUT
		(* The width of the rectangle to set. *)
		width : LREAL;
		(* The height of the rectangle to set. *)
		height : LREAL;
	END_VAR
END_METHOD


	(* Get the area of the rectangle. *)
	METHOD GetArea : LREAL
END_METHOD


	PROPERTY width : LREAL
GET
END_GET
SET
END_SET
END_PROPERTY


	PROPERTY height : LREAL
GET
END_GET
SET
END_SET
END_PROPERTY

END_FUNCTION_BLOCK

// POUs/Shapes/Geometry3D/3D/Sphere3D

	{attribute 'c++_compatible'}
	{attribute 'external_name' := 'Sphere3D_GUID_8042695E_7F9E_9D30_F784_8355A5E4C01A'}
	{attribute 'TcIecLibraryType'}
	{attribute 'no_explicit_call' :='do not call this POU directly'}
	{attribute 'no_assign'}
	FUNCTION_BLOCK Sphere3D EXTENDS Geometry3D


	(* Internal method *)
	METHOD FB_init : BOOL
	VAR_INPUT
		(*  if TRUE, the retain variables are initialized (warm start / cold start) *)
		bInitRetains : BOOL;
		(*  if TRUE, the instance afterwards gets moved into the copy code (online change) *)
		bInCopyCode : BOOL;
	END_VAR
END_METHOD


	(* Internal method *)
	{attribute 'hide'}
	METHOD FB_exit : BOOL
	VAR_INPUT
		(*  if TRUE, the exit method is called for exiting an instance that is copied afterwards (online change). *)
		bInCopyCode : BOOL;
	END_VAR
END_METHOD


	(* Get the volume of the sphere. *)
	METHOD GetVolume : LREAL
END_METHOD


	PROPERTY radius : LREAL
GET
END_GET
SET
END_SET
END_PROPERTY

END_FUNCTION_BLOCK

// POUs/Shapes/Geometry3D/3D/Cuboid3D

	{attribute 'c++_compatible'}
	{attribute 'external_name' := 'Cuboid3D_GUID_7258FDDD_0A71_9B07_CDA3_5D8E943844B2'}
	{attribute 'TcIecLibraryType'}
	{attribute 'no_explicit_call' :='do not call this POU directly'}
	{attribute 'no_assign'}
	FUNCTION_BLOCK Cuboid3D EXTENDS Geometry3D


	(* Internal method *)
	METHOD FB_init : BOOL
	VAR_INPUT
		(* if TRUE, the retain variables are initialized (warm start / cold start) *)
		bInitRetains : BOOL;
		(* if TRUE, the instance afterwards gets moved into the copy code (online change) *)
		bInCopyCode : BOOL;
	END_VAR
END_METHOD


	(* Internal method *)
	{attribute 'hide'}
	METHOD FB_exit : BOOL
	VAR_INPUT
		(* if TRUE, the exit method is called for exiting an instance that is copied afterwards (online change). *)
		bInCopyCode : BOOL;
	END_VAR
END_METHOD


	(* Set the dimensions of the cuboid. *)
	METHOD SetDimensions
	VAR_INPUT
		(* local x-component *)
		length : LREAL;
		(* local y-component *)
		width : LREAL;
		(* local z-component *)
		height : LREAL;
	END_VAR
END_METHOD


	(* Get the volume of the cuboid. *)
	METHOD GetVolume : LREAL
END_METHOD


	PROPERTY length : LREAL
GET
END_GET
SET
END_SET
END_PROPERTY


	PROPERTY width : LREAL
GET
END_GET
SET
END_SET
END_PROPERTY


	PROPERTY height : LREAL
GET
END_GET
SET
END_SET
END_PROPERTY

END_FUNCTION_BLOCK

// POUs/Shapes/Geometry3D/3D/Cylinder3D

	{attribute 'c++_compatible'}
	{attribute 'external_name' := 'Cylinder3D_GUID_16C6A7E7_2D59_93E5_D3F0_E345B5901415'}
	{attribute 'TcIecLibraryType'}
	{attribute 'no_explicit_call' :='do not call this POU directly'}
	{attribute 'no_assign'}
	FUNCTION_BLOCK Cylinder3D EXTENDS Geometry3D


	(* Internal method *)
	METHOD FB_init : BOOL
	VAR_INPUT
		(* if TRUE, the retain variables are initialized (warm start / cold start) *)
		bInitRetains : BOOL;
		(* if TRUE, the instance afterwards gets moved into the copy code (online change) *)
		bInCopyCode : BOOL;
	END_VAR
END_METHOD


	(* Internal method *)
	{attribute 'hide'}
	METHOD FB_exit : BOOL
	VAR_INPUT
		(* if TRUE, the exit method is called for exiting an instance that is copied afterwards (online change). *)
		bInCopyCode : BOOL;
	END_VAR
END_METHOD


	(* Set the dimensions of the cylinder. *)
	METHOD SetDimensions
	VAR_INPUT
		(* The radius to set. *)
		radius : LREAL;
		(* The height to set. *)
		height : LREAL;
	END_VAR
END_METHOD


	(* Get the volume of the cylinder. *)
	METHOD GetVolume : LREAL
END_METHOD


	PROPERTY radius : LREAL
GET
END_GET
SET
END_SET
END_PROPERTY


	PROPERTY height : LREAL
GET
END_GET
SET
END_SET
END_PROPERTY

END_FUNCTION_BLOCK

// POUs/Shapes/Geometry3D/Functions/CheckCollision3D

	{attribute 'TcIecLibraryType'}
	{attribute 'external_name' := 'CheckCollision3D_GUID_7526A54C_4125_92DA_E85F_E30F35EB6E80'}
	(* Check if two geometries are currently colliding. *)
	FUNCTION CheckCollision3D : BOOL
	VAR_IN_OUT
		geometry0	:	IPlcGeometry3D;	(* 1st input geometry to check for collision. *)
		geometry1	:	IPlcGeometry3D;	(* 2nd input geometry to check of collision. *)
	END_VAR

END_FUNCTION

// POUs/Shapes/Geometry3D/Functions/GetDistance3D

	{attribute 'TcIecLibraryType'}
	{attribute 'external_name' := 'GetDistance3D_GUID_869F9B59_D6FF_95DE_C768_335789473B38'}
	(* Get the distance between two geometries. *)
	FUNCTION GetDistance3D : LREAL
	VAR_IN_OUT
		geometry0	:	IPlcGeometry3D;	(* 1st input geometry to calculate the distance of. *)
		geometry1	:	IPlcGeometry3D;	(* 2nd input geometry to calculate the distance of. *)
	END_VAR

END_FUNCTION

// POUs/Shapes/Geometry3D/Functions/GetLinkingLine3D

	{attribute 'TcIecLibraryType'}
	{attribute 'external_name' := 'GetLinkingLine3D_GUID_E5A29052_5630_9A0A_F4A5_5AC169DB10FA'}
	(* Get the shortest path between two geometries. *)
	FUNCTION GetLinkingLine3D : BOOL
	VAR_IN_OUT
		geometry0	:	IPlcGeometry3D;	(* 1st input geometry to calculate the linking line for. *)
		geometry1	:	IPlcGeometry3D;	(* 2nd input geometry to calculate the linking line for. *)
		linkingLine	:	Segment3D;	(* Return the resulting linking line. *)
	END_VAR

END_FUNCTION

// POUs/Shapes/Geometry3D/Functions/CreateIntersection2D

	{attribute 'TcIecLibraryType'}
	{attribute 'external_name' := 'CreateIntersection2D_GUID_D97F08BF_A10C_9172_EB8B_B7697692777E'}
	(* Create a collection of intersections along a plane definition. *)
	FUNCTION CreateIntersection2D : BOOL
	VAR_IN_OUT
		container3D	:	Container3D;	(* Input container to create the intersections of. *)
		planeFrame	:	PositionSE3;	(* The coordinate frame to indicate the origin of the plane. *)
		container2D	:	Container2D;	(* Return the resulting collection of intersection. *)
	END_VAR

END_FUNCTION
